// TIA Portal project "Pivot Arm" (V16)
// Vorlageprojekt für das Buch mit Zielsystem S7-1200

(* hardware
DEVICE "S7-1200-Station_1"  S7-1200 Station
   slot 0: "Baugruppenträger_0"  Rack  V1.0
   slot 1: "PLC_1"  CPU 1211C DC/DC/DC  6ES7 211-1AE40-0XB0  V4.1
*)

// ===== PLC "PLC_1"  CPU 1211C DC/DC/DC =====

VAR_GLOBAL   // PLC tag table "Standard-Variablentabelle"
   "start button(1)" AT %I0.0 : Bool;
   "stop button" AT %I10.1 : Bool;
   "DiffuseSensor1" AT %I10.2 : Bool;
   "DiffuseSensor2" AT %I10.3 : Bool;
   "DiffuseSensor3" AT %I10.4 : Bool;
   "BeltConveor(6m)" AT %Q0.0 : Bool;
   "BeltConveor(4m)" AT %Q0.1 : Bool;
   "BeltConveor(2m)" AT %Q0.2 : Bool;
   "PivotArmSorterTurn" AT %Q0.3 : Bool;
   "PivotArmSorter1Belt(+)" AT %Q0.4 : Bool;
   "StartButton(Light)" AT %Q0.5 : Bool;
   "StopButton(Light)" AT %Q0.6 : Bool;
   "Belt 6m" AT %Q5.0 : Bool;
   "start button" AT %I5.0 : Bool;
   "stop" AT %I5.1 : Bool;
   "Belt 2m" AT %Q5.1 : Bool;
   "sensor1" AT %I5.2 : Bool;
   "pivot  +" AT %Q5.3 : Bool;
   "sensor2" AT %I5.3 : Bool;
   "pivot turn" AT %Q5.2 : Bool;
   "belt 4m" AT %Q5.4 : Bool;
   "sensor3" AT %I5.4 : Bool;
   "start Indicator" AT %Q5.5 : Bool;
   "stop Indicator" AT %Q5.6 : Bool;
   "Tag_1" AT %M0.0 : Bool;
END_VAR

FUNCTION "MHJ-PLC-Lab-Function-S71200" : Void   // FC9000, SCL
{ S7_Optimized_Access := 'TRUE' }
VERSION : 0.1
   VAR_TEMP
      rdTimeReturn : Int;
      outputTime : DTL;
      SyncVal : Byte;
      forVal : Int;
      forVal_2 : Int;
      Value : Byte;
   END_VAR
   VAR CONSTANT
      CompVal : Byte := 16#34;
      Value_01 : Byte := 16#11;
      Value_01_DW : DWord := 16#A165_D992;
      Value_02_DW : DWord := 16#58BE_4401;
   END_VAR
BEGIN

   #Value:=PEEK(area := 16#82,
        dbNumber := 0,
        byteOffset := 511);
   #Value := #Value + 1;

   POKE(area := 16#82,
        dbNumber := 0,
        byteOffset := 511,
        value := #Value);

   POKE(area:=16#81,
        dbNumber:=0,
        byteOffset:=1016,
        value:=#Value_01_DW);
   POKE(area := 16#81,
        dbNumber := 0,
        byteOffset := 1020,
        value := #Value_02_DW);

   POKE(area := 16#81,
        dbNumber := 0,
        byteOffset := 511,
        value := B#16#00);

   FOR #forVal := 0 TO 120 DO
       FOR #forVal_2:=0 TO 10 DO
           #rdTimeReturn:=RD_SYS_T(#outputTime);
           #rdTimeReturn := WR_SYS_T(#outputTime);
           #rdTimeReturn := RD_SYS_T(#outputTime);
           #rdTimeReturn := WR_SYS_T(#outputTime);
       END_FOR;
       #SyncVal:= PEEK(area := 16#81,
                      dbNumber := 0,
                      byteOffset := 511);
       IF #SyncVal = #CompVal THEN
          GOTO M_1;
       END_IF;
   END_FOR;
   RETURN;

   M_1:
   POKE(area := 16#81,
        dbNumber := 0,
        byteOffset := 511,
        value := B#16#0);
END_FUNCTION

ORGANIZATION_BLOCK "Main"   // OB1, LAD, ProgramCycle
TITLE = "Main Program Sweep (Cycle)"
{ S7_Optimized_Access := 'TRUE' }
VERSION : 0.1
   VAR_INPUT
      Initial_Call : Bool;   // Initial call of this OB
      Remanence : Bool;   // =True, if remanent data are available
   END_VAR
BEGIN

REGION Network 1: Konnektierungsbaustein für PLC-Lab
   // Im Netzwerk 1 wird der Konnektierungsbaustein für PLC-Lab aufgerufen.
   // Dieser Aufruf darf nicht entfernt werden!
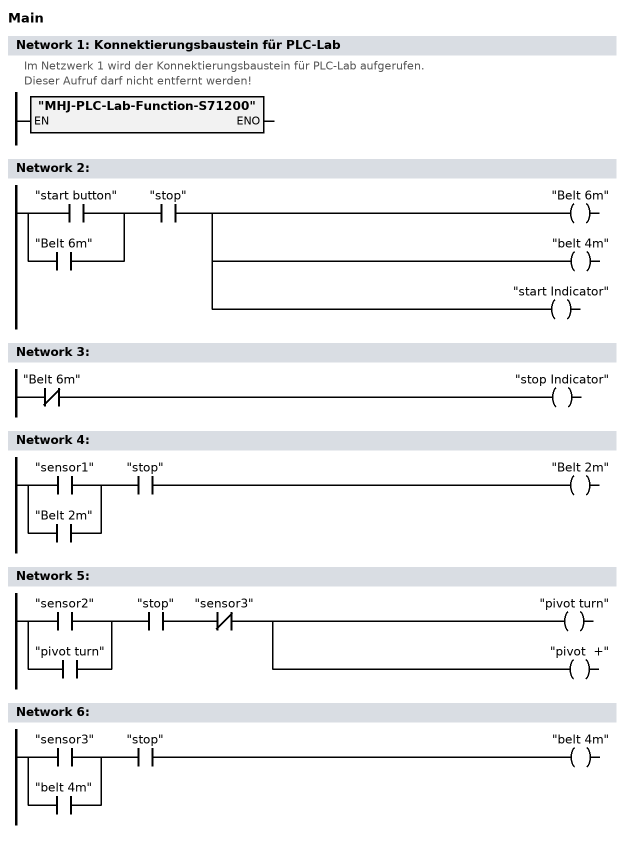
   RUNG wire#powerrail
      "MHJ-PLC-Lab-Function-S71200"()
   END_RUNG
   // the same network as SCL:
   "MHJ-PLC-Lab-Function-S71200"();
END_REGION

REGION Network 2
   RUNG wire#powerrail
      Contact( "start button" )
      wire#w1
      Contact( "stop" )
      wire#w2
      Coil( "Belt 6m" )
   END_RUNG
   RUNG wire#powerrail
      Contact( "Belt 6m" )
   END_RUNG wire#w1
   RUNG wire#w2
      Coil( "belt 4m" )
   END_RUNG
   RUNG wire#w2
      Coil( "start Indicator" )
   END_RUNG
   // the same network as SCL:
   "Belt 6m" := ("start button" OR "Belt 6m") AND "stop";
   "belt 4m" := "Belt 6m";
   "start Indicator" := "Belt 6m";
END_REGION

REGION Network 3
   RUNG wire#powerrail
      I_Contact( "Belt 6m" )
      Coil( "stop Indicator" )
   END_RUNG
   // the same network as SCL:
   "stop Indicator" := NOT "Belt 6m";
END_REGION

REGION Network 4
   RUNG wire#powerrail
      Contact( "sensor1" )
      wire#w1
      Contact( "stop" )
      Coil( "Belt 2m" )
   END_RUNG
   RUNG wire#powerrail
      Contact( "Belt 2m" )
   END_RUNG wire#w1
   // the same network as SCL:
   "Belt 2m" := ("sensor1" OR "Belt 2m") AND "stop";
END_REGION

REGION Network 5
   RUNG wire#powerrail
      Contact( "sensor2" )
      wire#w1
      Contact( "stop" )
      I_Contact( "sensor3" )
      wire#w2
      Coil( "pivot turn" )
   END_RUNG
   RUNG wire#powerrail
      Contact( "pivot turn" )
   END_RUNG wire#w1
   RUNG wire#w2
      Coil( "pivot  +" )
   END_RUNG
   // the same network as SCL:
   "pivot turn" := ("sensor2" OR "pivot turn") AND "stop" AND NOT "sensor3";
   "pivot  +" := "pivot turn";
END_REGION

REGION Network 6
   RUNG wire#powerrail
      Contact( "sensor3" )
      wire#w1
      Contact( "stop" )
      Coil( "belt 4m" )
   END_RUNG
   RUNG wire#powerrail
      Contact( "belt 4m" )
   END_RUNG wire#w1
   // the same network as SCL:
   "belt 4m" := ("sensor3" OR "belt 4m") AND "stop";
END_REGION
END_ORGANIZATION_BLOCK